# EPICS autosave request: iocs/merlinIOC/iocBoot/iocMerlin/auto_settings.req
file "medipix_settings.req",      P=$(P),  R=cam1:
file "NDStdArrays_settings.req",  P=$(P),  R=image1:
file "commonPlugin_settings.req", P=$(P)
